{attribute 'GeneratedUsingTerminal: EL1258-0000-0016'}
{attribute addProperty BoxType "EL1258-0000-0016"}
{attribute addProperty Id "Input_buffer_resetBOOL1Input_order_counterUSINT1"}
{attribute addProperty CRC "4053707553"}
{attribute addProperty Size "2"}
TYPE Ctrl_F19EAB21 :
STRUCT
	{attribute addProperty Name "Input_buffer_reset"}
	Input_buffer_reset : BOOL;
	{attribute addProperty Name "Input_order_counter"}
	Input_order_counter : USINT;
END_STRUCT
END_TYPE

(* stored: Version 1.2.0.0, ProductVersion 3.1.4024.9
   DUT Ctrl_F19EAB21: Id {d33167ba-8ed3-4476-bac1-3fdb2bd2aa6c} *)
